(* CoDeSys 2.3 export: BATHROOM_PIETRO.EXP *)

(* POU Rooms/Bathroom_pietro, ST *)
FUNCTION_BLOCK  Bathroom_pietro
VAR
	mainLamp:OnOff;
	wallLamp:OnOff;

END_VAR
mainLamp(input:=B3_3a OR P9_1a, output => B1_1);
wallLamp(input:=B3_3b, output => B2_2);
END_FUNCTION_BLOCK
